// TIA Portal V20 export
TYPE "typeEm1CommandsJobInterface"
// stored: Access Published, Namespace Unit1
   STRUCT
      reqAutoSplice { ExternalWritable := 'False'} : Bool;
   END_STRUCT;
END_TYPE
